FUNCTION_BLOCK MQTT_PUBLISHER_V3
  {SET_ATTRIBUTE(OpcUa, POINT.ENDPOINT)}
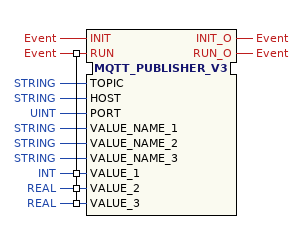
  EVENT_INPUT
    INIT;
    RUN WITH VALUE_1, VALUE_2, VALUE_3;
  END_EVENT
  EVENT_OUTPUT
    INIT_O;
    RUN_O;
  END_EVENT
  VAR_INPUT
    TOPIC : STRING; {SET_ATTRIBUTE(OpcUa, Constant)}
    HOST : STRING; {SET_ATTRIBUTE(OpcUa, Constant)}
    PORT : UINT; {SET_ATTRIBUTE(OpcUa, Constant)}
    VALUE_NAME_1 : STRING; {SET_ATTRIBUTE(OpcUa, Constant)}
    VALUE_NAME_2 : STRING; {SET_ATTRIBUTE(OpcUa, Constant)}
    VALUE_NAME_3 : STRING; {SET_ATTRIBUTE(OpcUa, Constant)}
    VALUE_1 : INT; {SET_ATTRIBUTE(OpcUa, Variable)}
    VALUE_2 : REAL; {SET_ATTRIBUTE(OpcUa, Variable)}
    VALUE_3 : REAL; {SET_ATTRIBUTE(OpcUa, Variable)}
  END_VAR
END_FUNCTION_BLOCK
